{attribute addProperty BoxType "EK1122-0000-0018"}
{attribute addProperty Id "boxessub_EK1100EK1100_179A0949162A_0030_EPP2339_0021_0016EPP2339_F1EE11F928836A_0031_EPP2339_0022_0016EPP2339_F1EE11F928836A_0032_EPP2349_0021_0016EPP2349_F1EE11F928836A_0033_EPP2349_0022_0016EPP2349_F1EE11F928836A_0034_EP2316_0008_0017EP2316_900F0E4A35244A_0035_EP2338_0001_0016EP2338_584B274D16020A_0036_EP2338_0001_0017EP2338_584B274D16020A_0037_EP2338_0002_0016EP2338_584B274D16020A_0038_EP2338_0002_0017EP2338_584B274D16020A_0039_EP2339_0021_0016EP2339_C622991433642A_0040_EP2339_0022_0016EP2339_EFDBABD528836"}
{attribute addProperty CRC "3284663404"}
{attribute addProperty SizeInBites "2784"}
{attribute addProperty SizeInBytes "348"}
TYPE boxesEK1122_C3C7FC6C EXTENDS EK1122_179A0949 :
STRUCT
	{attribute addProperty Name "boxessub_EK1100"}
	boxessub_EK1100 : EK1100_179A0949;
	{attribute addProperty Name "A_0030_EPP2339_0021_0016"}
	A_0030_EPP2339_0021_0016 : EPP2339_F1EE11F9;
	{attribute addProperty Name "A_0031_EPP2339_0022_0016"}
	A_0031_EPP2339_0022_0016 : EPP2339_F1EE11F9;
	{attribute addProperty Name "A_0032_EPP2349_0021_0016"}
	A_0032_EPP2349_0021_0016 : EPP2349_F1EE11F9;
	{attribute addProperty Name "A_0033_EPP2349_0022_0016"}
	A_0033_EPP2349_0022_0016 : EPP2349_F1EE11F9;
	{attribute addProperty Name "A_0034_EP2316_0008_0017"}
	A_0034_EP2316_0008_0017 : EP2316_900F0E4A;
	{attribute addProperty Name "A_0035_EP2338_0001_0016"}
	A_0035_EP2338_0001_0016 : EP2338_584B274D;
	{attribute addProperty Name "A_0036_EP2338_0001_0017"}
	A_0036_EP2338_0001_0017 : EP2338_584B274D;
	{attribute addProperty Name "A_0037_EP2338_0002_0016"}
	A_0037_EP2338_0002_0016 : EP2338_584B274D;
	{attribute addProperty Name "A_0038_EP2338_0002_0017"}
	A_0038_EP2338_0002_0017 : EP2338_584B274D;
	{attribute addProperty Name "A_0039_EP2339_0021_0016"}
	A_0039_EP2339_0021_0016 : EP2339_C6229914;
	{attribute addProperty Name "A_0040_EP2339_0022_0016"}
	A_0040_EP2339_0022_0016 : EP2339_EFDBABD5;
END_STRUCT
END_TYPE

(* stored: Version 1.2.0.0, ProductVersion 3.1.4024.9
   DUT boxesEK1122_C3C7FC6C: Id {13079dd0-d8bb-4982-93c0-f94e6ca56c74} *)
